FUNCTION_BLOCK XtsHardware EXTENDS CyclicBase IMPLEMENTS IXtsHardware, I_Initialise
VAR
	_Tracks : UDINT;
	_TmsSwitch : ITF_TmsSwitch;
	XtsIoEnvironment : Tc3_XTS_Utility.FB_TcIoXtsEnvironment;
	bInit: BOOL;
	bMoverIdDetectionError		: BOOL;
	bMoverIdDetectionActive		: BOOL;
	bMoverIdDetected : BOOL;
	f24V: ARRAY[1..SystemParameters.nModuleNumber] OF UINT;
	f48V: ARRAY[1..SystemParameters.nModuleNumber] OF UINT;
	CurrentLive : ARRAY[1..SystemParameters.nModuleNumber] OF DINT;
	MaxCurrent : ARRAY [1..SystemParameters.nModuleNumber] OF DINT;
	nModuleCounter : UINT := 1;
	i: UDINT;
	
	DetectedTracks : UDINT;
	DetectedModules : ARRAY[1..10] OF UDINT;
	PartIndex: UINT := 1;
	ModuleIndex : INT := 1;
	XtsHWInfo : XtsHardwareInfo;
	XtsHardwareOK : BOOL;
	bTriggerDetect: BOOL;
	
	DetectedParts: UDINT;
	Parts : ARRAY[1..SystemParameters.NumberOfParts] OF 
END_VAR

{analysis -2}

METHOD Cycle : HRESULT
VAR_INPUT
END_VAR
Cycle := S_OK;
IF NOT IsInSim() THEN
	getModuleInfoData();
END_IF
END_METHOD

METHOD FB_init : BOOL
VAR_INPUT
	bInitRetains : BOOL; // if TRUE, the retain variables are initialized (warm start / cold start)
	bInCopyCode : BOOL;  // if TRUE, the instance afterwards gets moved into the copy code (online change)
	XtsRunner : I_XtsRunner;
END_VAR
XtsRunner.AddComponent(THIS^);
END_METHOD

METHOD getAllMoversValid : BOOL
VAR_INPUT
END_VAR
 IF XtsIoEnvironment.XpuTcIo(1).GetAreAllPositionsValid() THEN
	 getAllMoversValid := TRUE;
	 Logger.Send(TC_EVENTS.XtsHardwareEvents.AllMoversValid,'');
 END_IF
END_METHOD

METHOD getModuleInfoData : BOOL
VAR_INPUT
END_VAR
IF XtsIoEnvironment.XpuTcIo(1).PartTcIo(PartIndex).ModuleCoE(nModuleCounter).InfoData.Update() THEN
	CurrentLive[ModuleIndex]:=XtsIoEnvironment.XpuTcIo(1).PartTcIo(PartIndex).ModuleCoE(nModuleCounter).InfoData.OverallCurrent;
	MaxCurrent[ModuleIndex]:=XtsIoEnvironment.XpuTcIo(1).PartTcIo(PartIndex).ModuleCoE(nModuleCounter).InfoData.MaxOverallCurrentLast500ms;
	f24V[ModuleIndex]:=XtsIoEnvironment.XpuTcIo(1).PartTcIo(PartIndex).ModuleCoE(nModuleCounter).InfoData.AuxiliaryVoltage24V;
	f48V[ModuleIndex]:=XtsIoEnvironment.XpuTcIo(1).PartTcIo(PartIndex).ModuleCoE(nModuleCounter).InfoData.DcLinkVoltage;
	ModuleIndex := ModuleIndex + 1;
	IF UINT_TO_UDINT(nModuleCounter) = DetectedModules[PartIndex] THEN
		nModuleCounter := 1;
		IF UINT_TO_UDINT(PartIndex) = DetectedParts THEN
			PartIndex := 1;
			ModuleIndex := 1;
		ELSE
			PartIndex := PartIndex + 1;
		END_IF
	ELSE
		nModuleCounter := nModuleCounter + 1;
	END_IF
END_IF
END_METHOD

METHOD PUBLIC GetMoverEnvInterface : I_TcIoXtsXpuMover
VAR_INPUT
	MoverNumber : UINT;
END_VAR
GetMoverEnvInterface := XtsIoEnvironment.XpuTcIo(1).MoverTcIo(MoverNumber);
END_METHOD

METHOD getMoversDetected : BOOL
VAR_INPUT
END_VAR
IF XtsIoEnvironment.XpuTcIo(1).GetDetectedMoverCount() = XtsIoEnvironment.XpuTcIo(1).GetExpectedMoverCount() THEN
	getMoversDetected := TRUE;
	Logger.Send(TC_EVENTS.XtsHardwareEvents.ExpectedMoversDetected,UDINT_TO_STRING(XtsIoEnvironment.XpuTcIo(1).GetExpectedMoverCount()));
ELSE
	getMoversDetected := FALSE;
	Logger.Send(TC_EVENTS.XtsHardwareEvents.ExpectedMoversNotFound,'');
END_IF
END_METHOD

METHOD PUBLIC GetTrackAssembly : BOOL
VAR_INPUT
END_VAR
DetectedTracks :=  XtsIoEnvironment.XpuTcIo(1).GetTrackCount();
IF DetectedTracks <> _Tracks THEN
	Logger.Send(TC_EVENTS.XtsHardwareEvents.XtsTracksCountError,'');
	RETURN; 
END_IF
DetectedParts := XtsIoEnvironment.XpuTcIo(1).GetPartCount();
FOR i := 1 TO DetectedParts DO
	DetectedModules[i] := XtsIoEnvironment.XpuTcIo(1).PartTcIo(UDINT_TO_UINT(i)).GetModuleCount();
END_FOR
GetTrackAssembly := TRUE;

XtsHWInfo.NoOfModules := DetectedModules;
XtsHWInfo.NoOfParts := DetectedParts;
XtsHWInfo.NoOfTracks := DetectedTracks;
END_METHOD

METHOD Initialise : HRESULT
VAR_INPUT
END_VAR
IF XtsIoEnvironment.Init(TRUE) THEN
	XtsIoEnvironment.Init(FALSE);
	Initialise := 2;
END_IF

XtsIoEnvironment.XpuTcIo(1).GetTrackOids();
END_METHOD

METHOD Is24VOK : HRESULT
VAR_INPUT
END_VAR
Is24VOK := 2;
FOR i := 1 TO UINT_TO_UDINT(SystemParameters.nModuleNumber) DO
	IF f24V[i] < 20400 THEN
		Is24VOK := 1;
	END_IF
	IF f24V[i] > 28800 THEN
		Is24VOK := 1;
	END_IF
END_FOR
END_METHOD

METHOD Is48VOK : HRESULT
VAR_INPUT
END_VAR
Is48VOK := 2;
FOR i := 1 TO UINT_TO_UDINT(SystemParameters.nModuleNumber) DO
	IF f48V[i] < 46080 THEN
		Is48VOK := 1;
	END_IF
	IF f48V[i] > 49920 THEN
		Is48VOK := 1;
	END_IF
END_FOR
END_METHOD

METHOD IsInSim : BOOL
VAR_INPUT
END_VAR
IF  XtsIoEnvironment.XpuTcIo(1).GetOperationMode() = OperationMode.Simulation THEN
	IsInSim := TRUE;
	Logger.Send(TC_EVENTS.XtsHardwareEvents.XtsInSimulationMode,'');
ELSE
	IsInSim := FALSE;
END_IF
END_METHOD

METHOD SetTracksForDetection : BOOL
VAR_INPUT
END_VAR
FOR i:=1 TO XtsIoEnvironment.XpuTcIo(1).GetTrackCount() DO
	XtsIoEnvironment.XpuTcIo(1).TrackTcIo(UDINT_TO_UINT(i)).SetIsIncludedInDetection(FALSE);
END_FOR

IF XtsIoEnvironment.XpuTcIo(1).GetTrackCount() = 1 THEN
	XtsIoEnvironment.XpuTcIo(1).TrackTcIo(1).SetIsIncludedInDetection(TRUE);
	Logger.Send(TC_EVENTS.XtsHardwareEvents.ActiveTracksAddedForDetection, UDINT_TO_STRING(XtsIoEnvironment.XpuTcIo(1).GetTrackCount()));
	SetTracksForDetection := TRUE;
ELSE
	SetTracksForDetection := TRUE;
	CASE _TmsSwitch.Switch OF
		TmsSwitchPosition.Up: 
			XtsIoEnvironment.XpuTcIo(1).TrackTcIo(3).SetIsIncludedInDetection(TRUE);
		TmsSwitchPosition.Middle:
			XtsIoEnvironment.XpuTcIo(1).TrackTcIo(1).SetIsIncludedInDetection(TRUE);
			XtsIoEnvironment.XpuTcIo(1).TrackTcIo(2).SetIsIncludedInDetection(TRUE);
		TmsSwitchPosition.Down:
			XtsIoEnvironment.XpuTcIo(1).TrackTcIo(4).SetIsIncludedInDetection(TRUE);
		ELSE
			SetTracksForDetection := FALSE;
	END_CASE
	Logger.Send(TC_EVENTS.XtsHardwareEvents.ActiveTracksAddedForDetection, UDINT_TO_STRING(XtsIoEnvironment.XpuTcIo(1).GetTrackCount()));
END_IF
END_METHOD

PROPERTY TmsSwitch : ITF_TmsSwitch
GET
TmsSwitch := _TmsSwitch;
END_GET
SET
_TmsSwitch := TmsSwitch;
END_SET
END_PROPERTY

PROPERTY Tracks : udint
GET
Tracks := _Tracks;
END_GET
SET
_Tracks	 := Tracks;
END_SET
END_PROPERTY

METHOD TriggerMoverDetection : BOOL
VAR_INPUT
END_VAR
XtsIoEnvironment.XpuTcIo(1).TriggerRedetection();
Logger.Send(TC_EVENTS.XtsHardwareEvents.MoverDetectionInitiated,'');
TriggerMoverDetection := true;
END_METHOD

METHOD TriggerMoverID : BOOL
VAR_INPUT
END_VAR
// Mover1 Functionality		
// Check if "MoverIdDetectionMode" has been activated under the XtsProcessingUnit object.
IF XtsIoEnvironment.XpuTcIo(1).GetMoverIdDetectionMode() = E_MoverIdDetectionMode.Mover1 THEN

	// Check if the "MoverIdDetection" has already been started or the Mover1 was found.
	IF NOT (bMoverIdDetectionActive OR bMoverIdDetected OR bTriggerDetect) THEN
		// Trigger the "MoverIdDetection".
		XtsIoEnvironment.XpuTcIo(1).TriggerMoverIdDetection();
		Logger.Send(TC_EVENTS.XtsHardwareEvents.Mover1DetectionStarted,'');
		bTriggerDetect := true;
	END_IF

	// Check for error or success of "MoverIdDetection".
	bMoverIdDetectionError 	:= XtsIoEnvironment.XpuTcIo(1).GetHasMoverIdDetectionError();
	bMoverIdDetected 	:= XtsIoEnvironment.XpuTcIo(1).GetIsMoverIdDetectionValid();
	bMoverIdDetectionActive	:= XtsIoEnvironment.XpuTcIo(1).GetIsMoverIdDetectionActive();
	
	// If the detection has an error, check for errors in output and try again.
	IF bMoverIdDetectionError THEN
		Logger.Send(TC_EVENTS.XtsHardwareEvents.Mover1DetectionFailed,'');
		RETURN; 
	END_IF

	// Do not process any further until the "MoverId" was deteced.
	IF NOT bMoverIdDetected THEN
		RETURN;
	END_IF	
	TriggerMoverID := TRUE;	
	Logger.Send(TC_EVENTS.XtsHardwareEvents.Mover1DetectionComplete,'');
ELSE
	TriggerMoverID := TRUE;
	Logger.Send(TC_EVENTS.XtsHardwareEvents.StandardMoverNumberingComplete,'');
END_IF
END_METHOD

END_FUNCTION_BLOCK

(* stored: Version 1.1.0.1, ProductVersion 3.1.4024.12
   POU XtsHardware: Id {01d7c7ee-eaba-4d97-9e2a-cab8b593df67}, SpecialFunc None
   Method Cycle: Id {b464f15b-ca99-474e-bc8b-11279972c349}
   Method FB_init: Id {7d0880e3-23ff-433e-9f1f-2df9860acb17}
   Method getAllMoversValid: Id {c4e70289-55ca-41b9-a3bc-195801ae93a3}
   Method getModuleInfoData: Id {3efa41b4-5489-4d81-8938-0f058eef3c58}
   Method GetMoverEnvInterface: Id {1fc643c6-ecb9-4760-af6a-4f21ce7c87e0}
   Method getMoversDetected: Id {5e49a15e-96a4-4ef0-90a8-d0eb7c5a7559}
   Method GetTrackAssembly: Id {ce747361-f640-4f49-a834-f6cbf088a32a}
   Method Initialise: Id {238260bf-972c-4836-891f-55586c0f1b1a}
   Method Is24VOK: Id {2b0cb545-a877-4023-acf7-204433c79109}
   Method Is48VOK: Id {85bd6738-1af1-443c-8d2c-d0704993fb05}
   Method IsInSim: Id {1d10bcec-acec-45d5-bf84-489041573d3d}
   Method SetTracksForDetection: Id {ddc7d054-a36f-42ec-9521-b7a91e617287}
   Property TmsSwitch: Id {3e77501e-8518-4e1c-97a5-5dc9bc6d0fd4}
   Get Get: Id {b0d03380-5fb6-4b27-9e19-7629ccd57ac3}
   Set Set: Id {ca7bb02b-1706-4344-953d-c58662955917}
   Property Tracks: Id {8efe48a8-9199-4a7a-a2ff-c779a3700ab7}
   Get Get: Id {e0b3b297-c3c4-4edc-8048-0ed07c7f0ba3}
   Set Set: Id {e5c09f87-cbe9-4bf0-ba07-78bfac777483}
   Method TriggerMoverDetection: Id {7ec0784a-bc20-43d5-9663-6bc83fb38f70}
   Method TriggerMoverID: Id {3caa48f4-4134-416c-8ece-2720f801ed03} *)
